FUNCTION_BLOCK FB_DataChannelRecvFifo EXTENDS FB_ArrayFifo
VAR
	m_pDataChannel: POINTER TO FB_DataChannelRecvBase;
	m_bolEnable: BOOL;
	m_intMaxFifoSize: INT := 10;
	m_pItem: POINTER TO BYTE;
	m_bolResult: BOOL;
END_VAR

(* Copyright 2017 Cimpress

Licensed under the Apache License, Version 2.0 (the "License");
you may not use this file except in compliance with the License.
You may obtain a copy of the License at

http://www.apache.org/licenses/LICENSE-2.0

Unless required by applicable law or agreed to in writing, software
distributed under the License is distributed on an "AS IS" BASIS,
WITHOUT WARRANTIES OR CONDITIONS OF ANY KIND, either express or implied.
See the License for the specific language governing permissions and
limitations under the License. *)

IF m_bolEnable AND (m_pItem <> Tc3_MemMan.NULL) THEN
	IF NOT m_pDataChannel^.Busy THEN
		m_bolResult := m_pDataChannel^.GetData(
						udiDataSize := m_pDataChannel^.DataSize,
						pData		:= m_pItem);

		IF m_uinItemCount < m_uinMaxItemCount THEN
			Push(m_pItem);
		ELSE
			m_pDataChannel^.Error := 1;
		END_IF 	
	END_IF
	
	m_pDataChannel^();
END_IF

PROPERTY Item : POINTER TO BYTE
GET
END_GET
SET
m_pItem := Item;
END_SET
END_PROPERTY

PROPERTY Enable : BOOL
GET
Enable := m_bolEnable;
END_GET
SET
m_bolEnable := Enable;
END_SET
END_PROPERTY

PROPERTY MaxFifoSize : INT
GET
MaxFifoSize := m_intMaxFifoSize;
END_GET
SET
m_intMaxFifoSize := MaxFifoSize;
END_SET
END_PROPERTY

PROPERTY DataChannel : POINTER TO FB_DataChannelRecvBase
SET
m_pDataChannel := DataChannel;
END_SET
END_PROPERTY

END_FUNCTION_BLOCK

(* stored: Version 1.1.0.1, ProductVersion 3.1.4019.2
   POU FB_DataChannelRecvFifo: Id {df3e4527-53f0-4710-9158-aa4780fb5da2}, SpecialFunc None
   Property Item: Id {2ad1ced4-8717-40a7-a67c-474c04794bc6}
   Get Get: Id {45600d03-4bea-4872-936e-b920000257d8}
   Set Set: Id {c127d49e-7e34-4fbb-8169-248801b04e2a}
   Property Enable: Id {ad58ea5f-4fdc-4c0d-9539-b6bc00c09646}
   Get Get: Id {12fcb4b6-ac53-4f4a-929b-c1c40a38e731}
   Set Set: Id {39deef12-6c42-4881-b72a-a6288f4056f8}
   Property MaxFifoSize: Id {d45af4a2-02a8-4699-8250-fe883089c076}
   Get Get: Id {202c6cb9-14bc-4c9f-8a62-4fb19c47be23}
   Set Set: Id {2a11508c-a9f7-4e91-9b06-cc1b2b5cc218}
   Property DataChannel: Id {f8936c45-1727-46ac-b706-a9cec4d851a8}
   Set Set: Id {c607b92d-1d39-449c-83ca-55ec034eef79} *)
